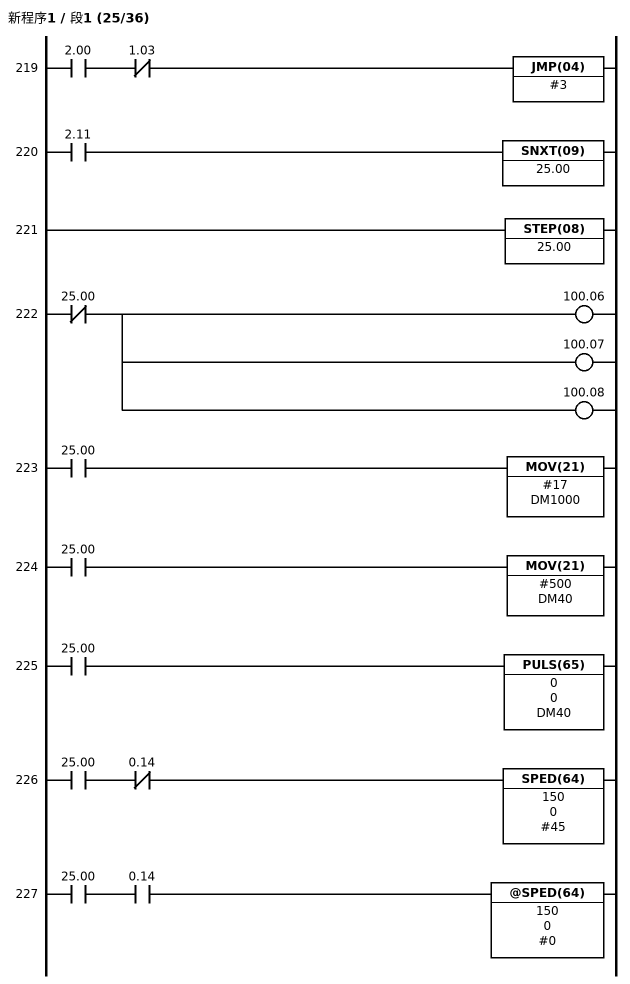
; [picture p24: 新程序1 / 段1, rungs 219-227]
; rung 219
LD 2.00
ANDNOT 1.03
JMP(04) #3
; rung 220
LD 2.11
SNXT(09) 25.00
; rung 221
STEP(08) 25.00
; rung 222
LDNOT 25.00
OUT 100.06
OUT 100.07
OUT 100.08
; rung 223
LD 25.00
MOV(21) #17 DM1000
; rung 224
LD 25.00
MOV(21) #500 DM40
; rung 225
LD 25.00
PULS(65) 0 0 DM40
; rung 226
LD 25.00
ANDNOT 0.14
SPED(64) 150 0 #45
; rung 227
LD 25.00
AND 0.14
@SPED(64) 150 0 #0

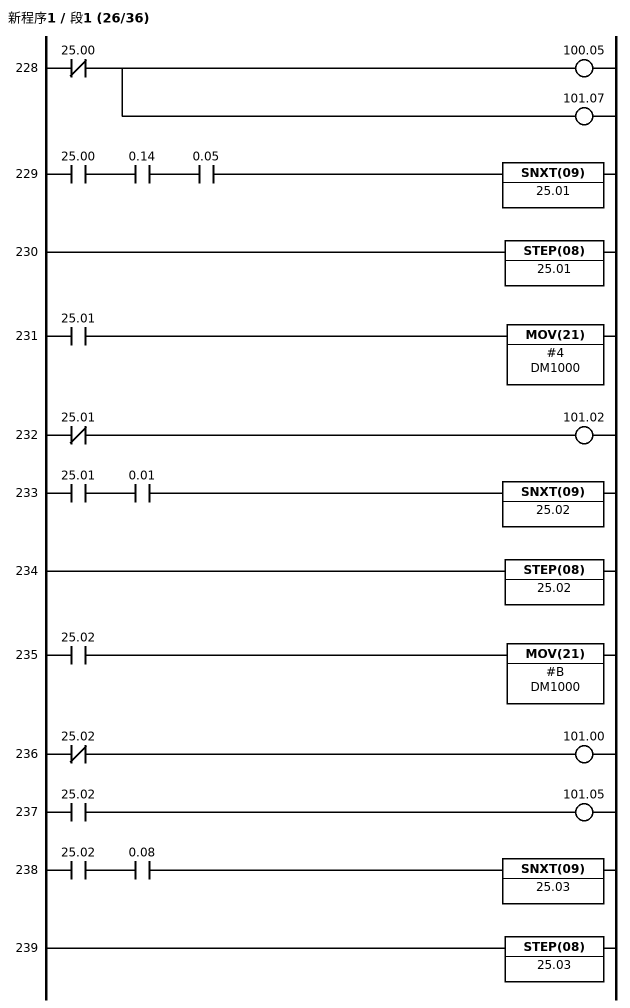
; rung 228
LDNOT 25.00
OUT 100.05
OUT 101.07
; rung 229
LD 25.00
AND 0.14
AND 0.05
SNXT(09) 25.01
; rung 230
STEP(08) 25.01
; rung 231
LD 25.01
MOV(21) #4 DM1000
; rung 232
LDNOT 25.01
OUT 101.02
; rung 233
LD 25.01
AND 0.01
SNXT(09) 25.02
; rung 234
STEP(08) 25.02
; rung 235
LD 25.02
MOV(21) #B DM1000
; rung 236
LDNOT 25.02
OUT 101.00
; rung 237
LD 25.02
OUT 101.05
; rung 238
LD 25.02
AND 0.08
SNXT(09) 25.03
; rung 239
STEP(08) 25.03

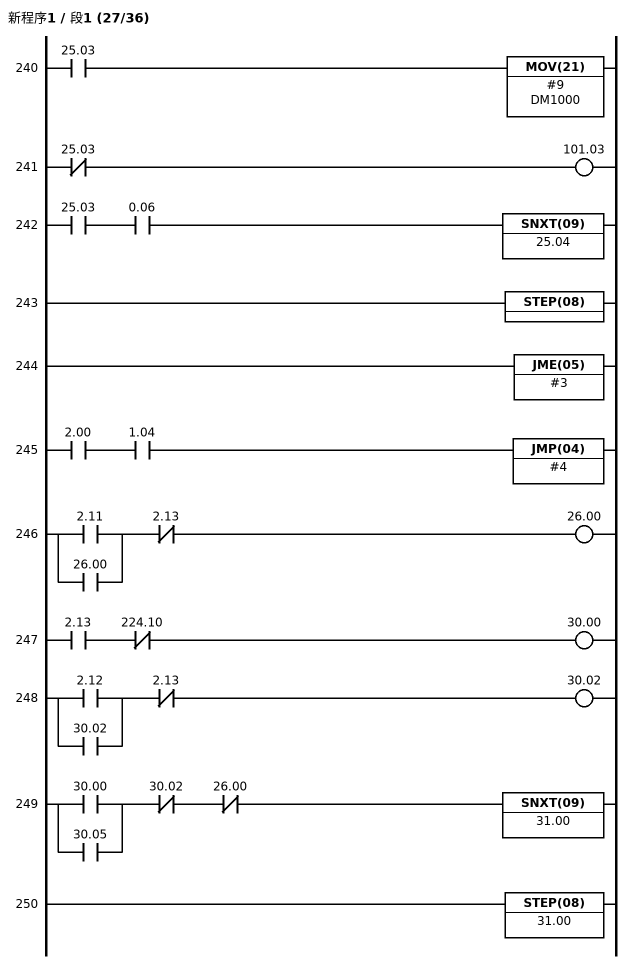
; rung 240
LD 25.03
MOV(21) #9 DM1000
; rung 241
LDNOT 25.03
OUT 101.03
; rung 242
LD 25.03
AND 0.06
SNXT(09) 25.04
; rung 243
STEP(08)
; rung 244
JME(05) #3
; rung 245
LD 2.00
AND 1.04
JMP(04) #4
; rung 246
LD 2.11
OR 26.00
ANDNOT 2.13
OUT 26.00
; rung 247
LD 2.13
ANDNOT 224.10
OUT 30.00
; rung 248
LD 2.12
OR 30.02
ANDNOT 2.13
OUT 30.02
; rung 249
LD 30.00
OR 30.05
ANDNOT 30.02
ANDNOT 26.00
SNXT(09) 31.00
; rung 250
STEP(08) 31.00

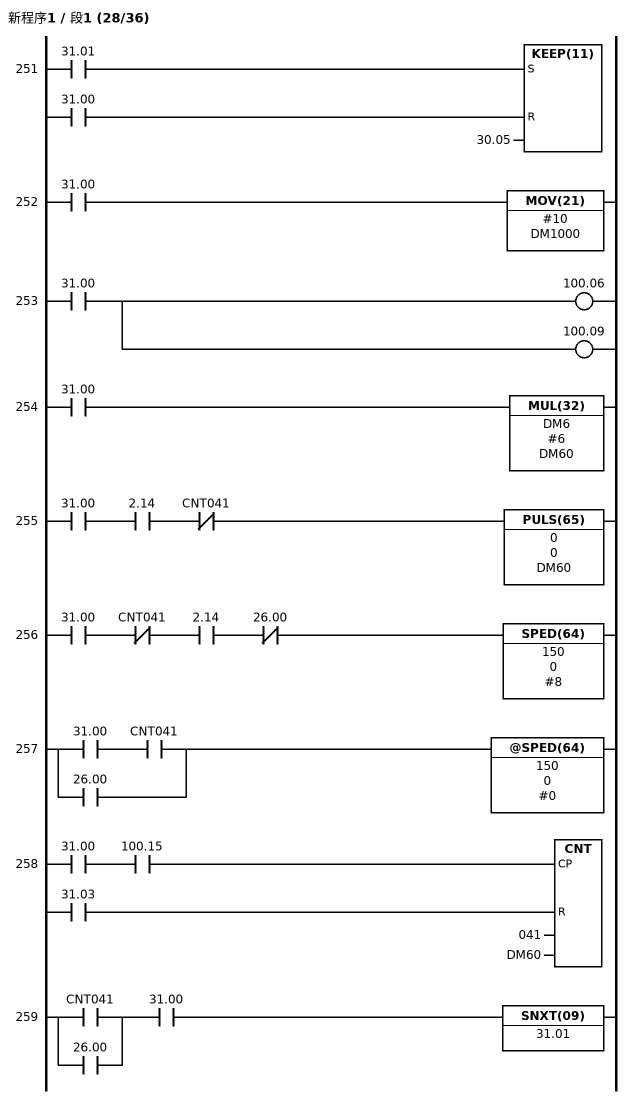
; rung 251
LD 31.01
LD 31.00
KEEP(11) 30.05
; rung 252
LD 31.00
MOV(21) #10 DM1000
; rung 253
LD 31.00
OUT 100.06
OUT 100.09
; rung 254
LD 31.00
MUL(32) DM6 #6 DM60
; rung 255
LD 31.00
AND 2.14
ANDNOT CNT041
PULS(65) 0 0 DM60
; rung 256
LD 31.00
ANDNOT CNT041
AND 2.14
ANDNOT 26.00
SPED(64) 150 0 #8
; rung 257
LD 31.00
AND CNT041
OR 26.00
@SPED(64) 150 0 #0
; rung 258
LD 31.00
AND 100.15
LD 31.03
CNT 041 DM60
; rung 259
LD CNT041
OR 26.00
AND 31.00
SNXT(09) 31.01

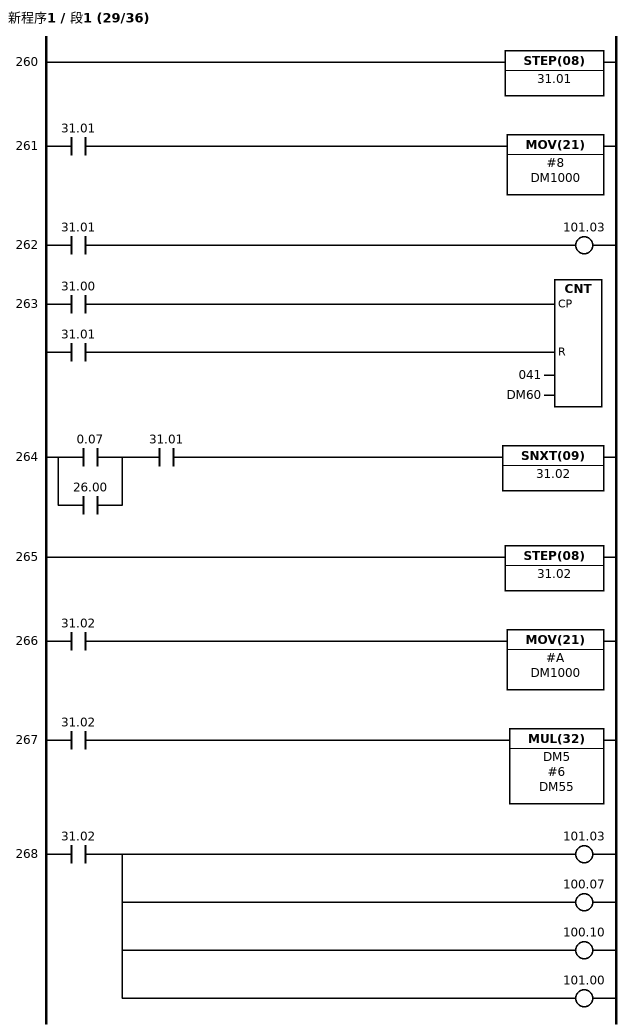
; rung 260
STEP(08) 31.01
; rung 261
LD 31.01
MOV(21) #8 DM1000
; rung 262
LD 31.01
OUT 101.03
; rung 263
LD 31.00
LD 31.01
CNT 041 DM60
; rung 264
LD 0.07
OR 26.00
AND 31.01
SNXT(09) 31.02
; rung 265
STEP(08) 31.02
; rung 266
LD 31.02
MOV(21) #A DM1000
; rung 267
LD 31.02
MUL(32) DM5 #6 DM55
; rung 268
LD 31.02
OUT 101.03
OUT 100.07
OUT 100.10
OUT 101.00

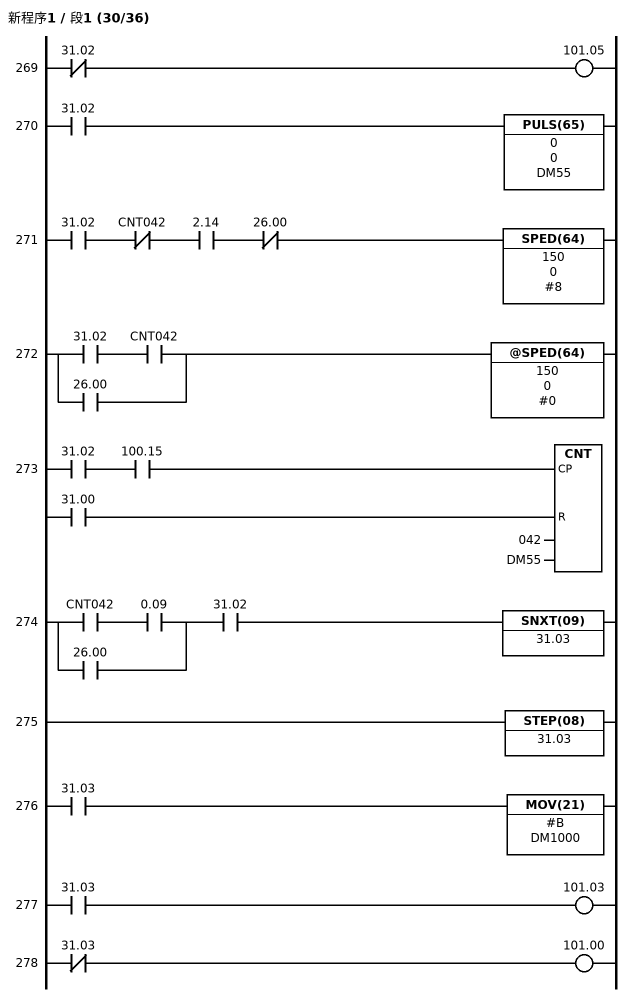
; rung 269
LDNOT 31.02
OUT 101.05
; rung 270
LD 31.02
PULS(65) 0 0 DM55
; rung 271
LD 31.02
ANDNOT CNT042
AND 2.14
ANDNOT 26.00
SPED(64) 150 0 #8
; rung 272
LD 31.02
AND CNT042
OR 26.00
@SPED(64) 150 0 #0
; rung 273
LD 31.02
AND 100.15
LD 31.00
CNT 042 DM55
; rung 274
LD CNT042
AND 0.09
OR 26.00
AND 31.02
SNXT(09) 31.03
; rung 275
STEP(08) 31.03
; rung 276
LD 31.03
MOV(21) #B DM1000
; rung 277
LD 31.03
OUT 101.03
; rung 278
LDNOT 31.03
OUT 101.00

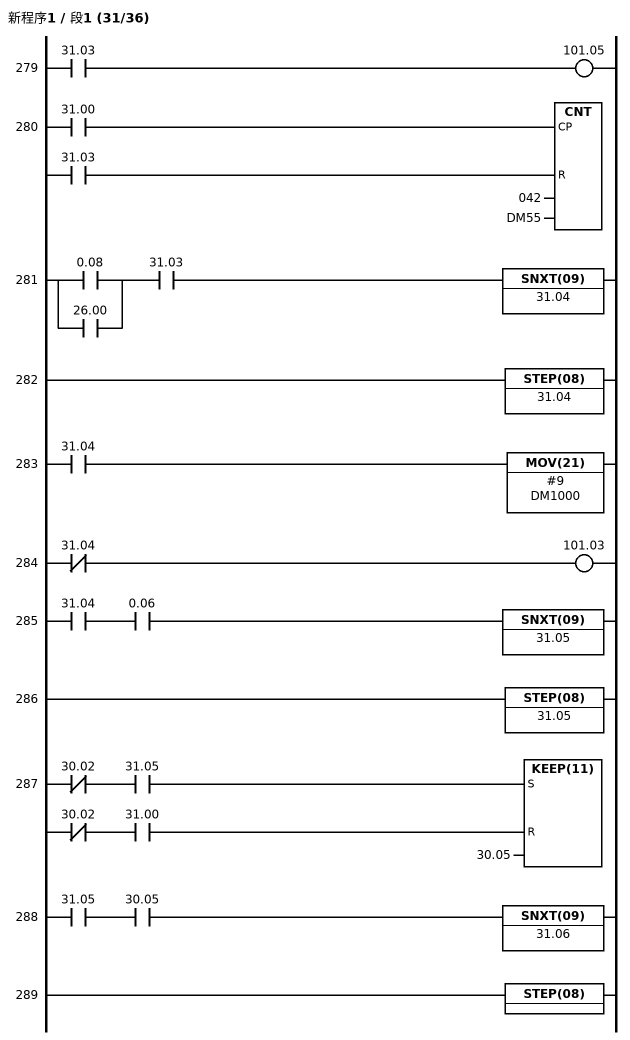
; rung 279
LD 31.03
OUT 101.05
; rung 280
LD 31.00
LD 31.03
CNT 042 DM55
; rung 281
LD 0.08
OR 26.00
AND 31.03
SNXT(09) 31.04
; rung 282
STEP(08) 31.04
; rung 283
LD 31.04
MOV(21) #9 DM1000
; rung 284
LDNOT 31.04
OUT 101.03
; rung 285
LD 31.04
AND 0.06
SNXT(09) 31.05
; rung 286
STEP(08) 31.05
; rung 287
LDNOT 30.02
AND 31.05
LDNOT 30.02
AND 31.00
KEEP(11) 30.05
; rung 288
LD 31.05
AND 30.05
SNXT(09) 31.06
; rung 289
STEP(08)

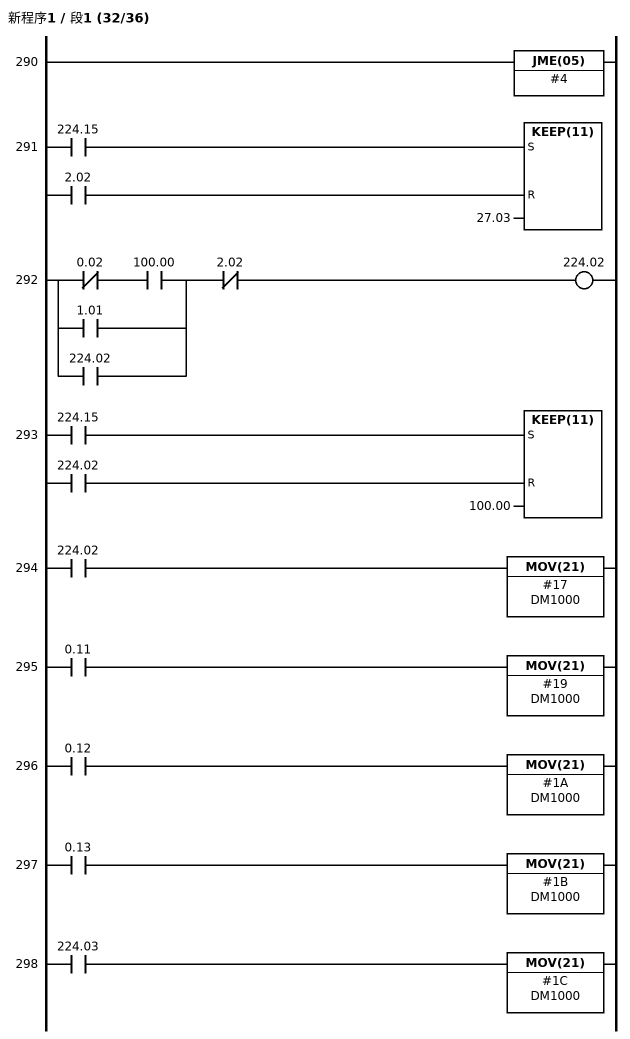
; rung 290
JME(05) #4
; rung 291
LD 224.15
LD 2.02
KEEP(11) 27.03
; rung 292
LDNOT 0.02
AND 100.00
OR 1.01
OR 224.02
ANDNOT 2.02
OUT 224.02
; rung 293
LD 224.15
LD 224.02
KEEP(11) 100.00
; rung 294
LD 224.02
MOV(21) #17 DM1000
; rung 295
LD 0.11
MOV(21) #19 DM1000
; rung 296
LD 0.12
MOV(21) #1A DM1000
; rung 297
LD 0.13
MOV(21) #1B DM1000
; rung 298
LD 224.03
MOV(21) #1C DM1000

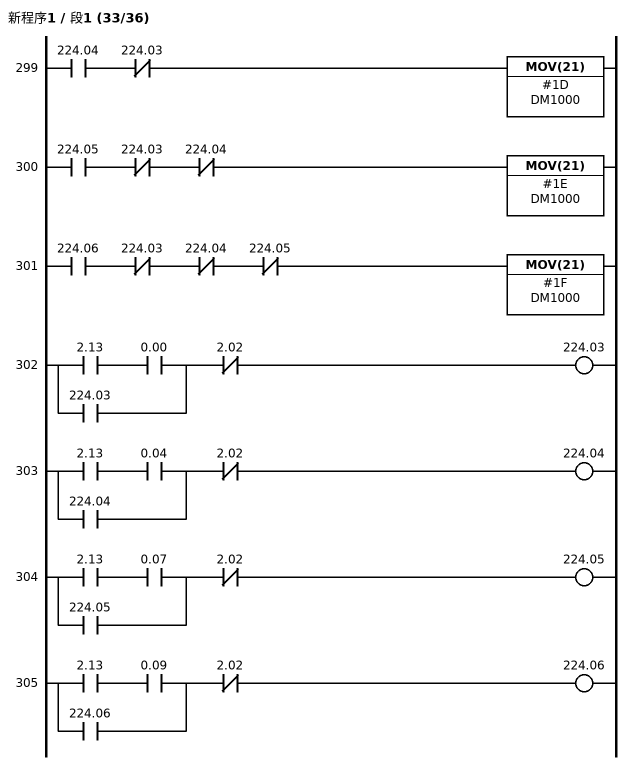
; rung 299
LD 224.04
ANDNOT 224.03
MOV(21) #1D DM1000
; rung 300
LD 224.05
ANDNOT 224.03
ANDNOT 224.04
MOV(21) #1E DM1000
; rung 301
LD 224.06
ANDNOT 224.03
ANDNOT 224.04
ANDNOT 224.05
MOV(21) #1F DM1000
; rung 302
LD 2.13
AND 0.00
OR 224.03
ANDNOT 2.02
OUT 224.03
; rung 303
LD 2.13
AND 0.04
OR 224.04
ANDNOT 2.02
OUT 224.04
; rung 304
LD 2.13
AND 0.07
OR 224.05
ANDNOT 2.02
OUT 224.05
; rung 305
LD 2.13
AND 0.09
OR 224.06
ANDNOT 2.02
OUT 224.06

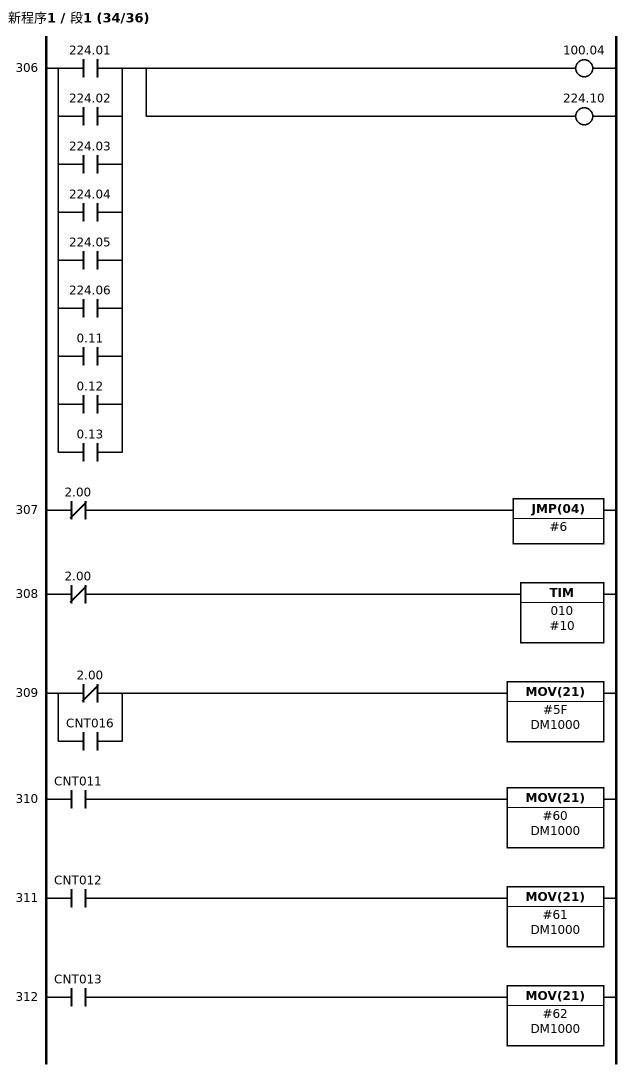
; rung 306
LD 224.01
OR 224.02
OR 224.03
OR 224.04
OR 224.05
OR 224.06
OR 0.11
OR 0.12
OR 0.13
OUT 100.04
OUT 224.10
; rung 307
LDNOT 2.00
JMP(04) #6
; rung 308
LDNOT 2.00
TIM 010 #10
; rung 309
LDNOT 2.00
OR CNT016
MOV(21) #5F DM1000
; rung 310
LD CNT011
MOV(21) #60 DM1000
; rung 311
LD CNT012
MOV(21) #61 DM1000
; rung 312
LD CNT013
MOV(21) #62 DM1000

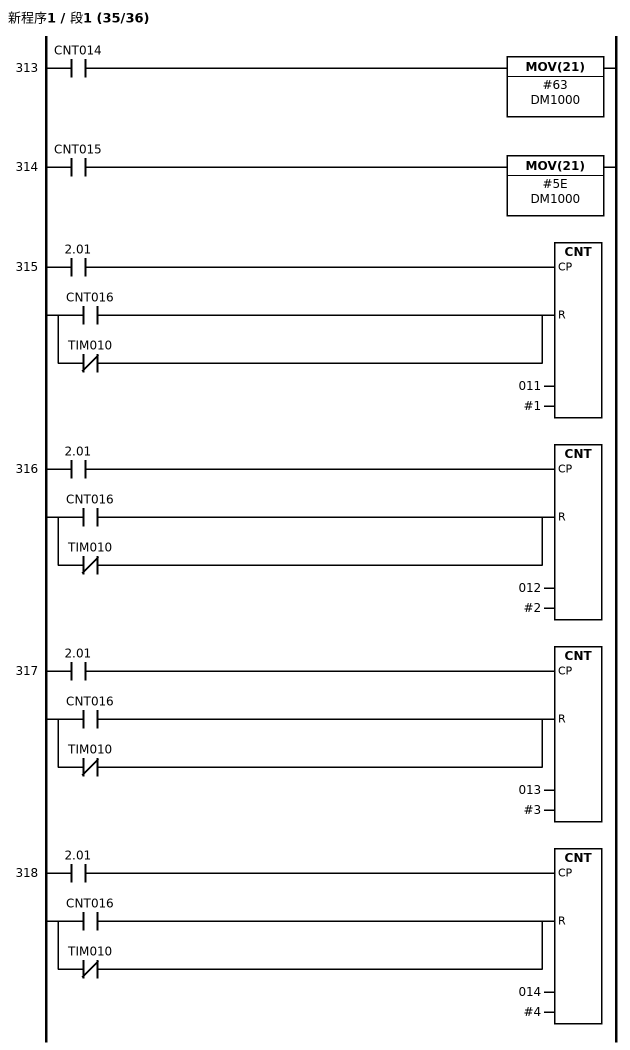
; rung 313
LD CNT014
MOV(21) #63 DM1000
; rung 314
LD CNT015
MOV(21) #5E DM1000
; rung 315
LD 2.01
LD CNT016
ORNOT TIM010
CNT 011 #1
; rung 316
LD 2.01
LD CNT016
ORNOT TIM010
CNT 012 #2
; rung 317
LD 2.01
LD CNT016
ORNOT TIM010
CNT 013 #3
; rung 318
LD 2.01
LD CNT016
ORNOT TIM010
CNT 014 #4

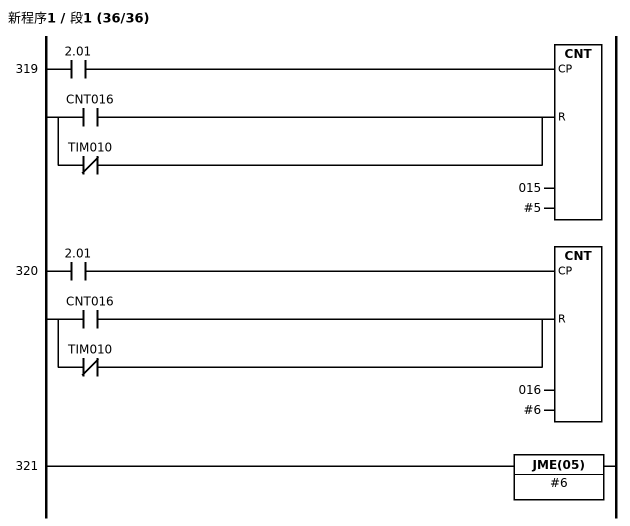
; rung 319
LD 2.01
LD CNT016
ORNOT TIM010
CNT 015 #5
; rung 320
LD 2.01
LD CNT016
ORNOT TIM010
CNT 016 #6
; rung 321
JME(05) #6
; rung 322
END(01)